(*

	
*)

FUNCTION_BLOCK RecordSQL IMPLEMENTS IRecordDB
VAR_INPUT
	nDBID						: UDINT;					// Database ID for TF6420
	DB_Parameter				: Tc2_Utilities.T_Arg;
END_VAR
VAR_OUTPUT
	bBusy			: BOOL;	// In writing database
	bError			: BOOL; // Somthing wrong situation happend
	TcResult		: Tc3_Database.I_TcMessage; // Response message
    sErrorMessage	: STRING(255);	// Error message
END_VAR
VAR
	
	//for generating timestamp
	fbGetSystemTime1: GetSystemTime;
	dwTimeLoDW: DWORD;
	dwTimeHiDW: DWORD;
	tFileTime: T_FILETIME;
	nTimestamp: LINT;
	
	//for insert samples
	fbPLCDBCmd: FB_PLCDBCmdEvt(sNetID := '', tTimeout := T#19S);

	// Variables for queue feature
	get_data 			: ChunkCommand;
	State				: E_DbLogState;
	_dbid				: UDINT;
	_queue 				: dequeue;	
	_query				: T_MaxString;
END_VAR


CASE State OF

	E_DbLogState.idle:
		
		IF NOT fbPLCDBCmd.bBusy THEN
			State := E_DbLogState.init;
		END_IF

	E_DbLogState.init:
	
		IF NOT fbPLCDBCmd.bBusy AND _queue.queue_usage > 0 THEN
			// getting data
			get_data := _queue.get();
			_query := get_data.sql_parameters.insert_query_string;
			State := E_DbLogState.writing;
		END_IF

	E_DbLogState.writing:
		//Write buffer element to database
		IF fbPLCDBCmd.Execute(nDBID, 
							ADR(_query), 
							SIZEOF(_query), 
							get_data.start_pointer, 
							get_data.structure_size * get_data.chunk_size, 
							get_data.sql_parameters.pParameters, 
							get_data.sql_parameters.cbParameters) THEN
			IF fbPLCDBCmd.bError THEN
				State := E_DbLogState.error;
			ELSE
				State := E_DbLogState.init;
			END_IF				
		END_IF
		

	E_DbLogState.error:
		//IF TcResult.RequestEventText(1033, sErrorMessage, SIZEOF(sErrorMessage)) THEN
            //TcResult.Send(F_GetSystemTime());
            State := E_DbLogState.idle;
            bError := TRUE;
        //END_IF

END_CASE

{warning 'add method implementation '}
METHOD FB_init : BOOL
VAR_INPUT
	(* if TRUE, the retain variables are initialized (warm start / cold start)*)
	bInitRetains	: BOOL;
	(* if TRUE, the instance afterwards gets moved into the copy code (online change)*)
	bInCopyCode	: BOOL;
	(*Database ID for TF6420 configurator*)
	DBID	: UDINT;
END_VAR
_dbid := DBID;
END_METHOD

{warning 'add property implementation'}
PROPERTY queue : REFERENCE TO dequeue
GET
queue REF= _queue;
END_GET
SET
_queue := queue;
END_SET
END_PROPERTY

END_FUNCTION_BLOCK

(* stored: Version 1.1.0.1, ProductVersion 3.1.4024.12
   POU RecordSQL: Id {c22ca813-56d1-45d3-a2ad-9ac2c556a6da}, SpecialFunc None
   Method FB_init: Id {f9b530cb-dfd9-430f-9dfa-fe8fa0d8029d}
   Property queue: Id {783f7123-f13b-436b-999f-bb0882697016}
   Get Get: Id {3aa55314-d948-4540-a239-89938f2bca68}
   Set Set: Id {5f8801a8-0e9c-4465-a8c8-048a23cf83b3} *)
